Fanuc KAREL source: kt00940.KL

PROGRAM KT00940
%STACKSIZE=65535
%PRIORITY=65535
%NOLOCKGROUP
VAR
ENTRY : INTEGER
PNAME : STRING[80]
VNAME : STRING[80]
STATUS : INTEGER
VALUE : XYZWPR
BEGIN
ENTRY=0
PNAME=''
VNAME='VALUE'
-- UNRESOLVED_PC line 13 opcodes [27 22 22 2A 22 2A 22 1C 22 AF] marker_code=43
END KT00940
